{attribute 'obsolete' := 'Use E_MotionFFType'}
TYPE ENUM_MotionFFType : E_MotionFFType; END_TYPE

(* stored: Version 1.1.0.1
   DUT ENUM_MotionFFType: Id {201ee7d6-ca7b-43e5-a41f-a1d695a8daec} *)
